// TwinCAT 3 PLC project Regions
// ProgramVersion: 3.1.4026.18
// libraries:
//   Tc3_Module, * (Beckhoff Automation GmbH)
//   ZApplication, 1.5.37.1 (Zeugwerk GmbH)
//   ZAux, 1.5.37.1 (Zeugwerk GmbH)
//   ZCore, 1.5.37.1 (Zeugwerk GmbH)
//   ZEquipment, 1.5.37.1 (Zeugwerk GmbH)
//   ZPlatform, 1.5.37.1 (Zeugwerk GmbH)
// project tree:
//   ZApp/App/ ZApp.TcPOU
//   ZApp/App/_DataTypes/ ZAppStep.TcDUT
//   ZApp/App/_States/ ZAppSequenceBoot.TcPOU, ZAppSequenceBootFault.TcPOU, ZAppSequenceRunning.TcPOU
//   ZApp/App/_SubObjects/ ZAppSequence.TcPOU
//   ZApp/Com/_DataTypes/ ZCom.TcDUT, ZComUnit.TcDUT
//   ZApp/Data/_DataTypes/ ZData.TcDUT, ZDataMachine.TcDUT, ZDataConfig.TcDUT, ZDataCalibration.TcDUT, ZDataRecipe.TcDUT
//   ZApp/SharedContext/ SharedContextCom.TcDUT, SharedContextComPublish.TcDUT, SharedContextComSubscribe.TcDUT, SharedContextContainer.TcPOU
//   ZApp/Unit/Handling/ HandlingUnit.TcPOU, HandlingUnitProgram.TcPOU, IHandling.TcIO
//   ZApp/Unit/Handling/_Com/ HandlingCom.TcDUT, HandlingComPublish.TcDUT, HandlingComPublishEquipment.TcDUT, HandlingComRef.TcDUT, HandlingComRequest.TcDUT, HandlingComSubscribe.TcDUT, HandlingComSubscribeEquipment.TcDUT
//   ZApp/Unit/Handling/_DataTypes/ HandlingState.TcDUT, HandlingStep.TcDUT
//   ZApp/Unit/Handling/_Data/ HandlingDataCalibration.TcDUT, HandlingDataConfig.TcDUT, HandlingDataMachine.TcDUT, HandlingDataRef.TcDUT
//   ZApp/Unit/Handling/_Equipment/ HandlingActuator.TcPOU, HandlingAxis.TcPOU, HandlingEquipment.TcPOU, HandlingFieldbus.TcPOU, HandlingIo.TcPOU, HandlingLinkedUnit.TcPOU
//   ZApp/Unit/Handling/_States/ HandlingSequenceAutomatic.TcPOU, HandlingSequenceBoot.TcPOU, HandlingSequenceFaultReaction.TcPOU, HandlingSequenceGoHome.TcPOU, HandlingSequenceStop.TcPOU, IPathQuery.TcIO, IPathQuery2.TcIO, IPathQuery3.TcIO, Path1d.TcPOU
//   ZApp/Unit/Handling/_SubObjects/ HandlingContainer.TcPOU, HandlingSequence.TcPOU
//   ZApp/ ZGlobal.TcGVL, ZModuleProgram.TcPOU, ZModuleTask.TcTTO
// real-time tasks:
//   TASK ZModuleTask: cycle T#10ms, priority 20, ADS port 350

CONFIGURATION Regions
    RESOURCE PLC ON TwinCAT3
        TASK ZModuleTask(INTERVAL := T#10ms, PRIORITY := 20);
        PROGRAM ZModuleProgram WITH ZModuleTask : ZModuleProgram;
    END_RESOURCE
END_CONFIGURATION

// ---- ZApp/App/_DataTypes/ZAppStep.TcDUT
{attribute 'qualified_only'}
{attribute 'to_string'}
TYPE ZAppStep :
(
  Undefined := 0
  
  ,BootBegin
  ,BootLoadDefaultData
  ,BootEnd
  ,BootFaultBegin
  ,BootFaultEnd 
  ,RunningBegin
  ,RunningEnd   
);
END_TYPE

// ---- ZApp/Com/_DataTypes/ZCom.TcDUT
TYPE ZCom :
STRUCT
  // module context
  App : ZApplication.ApplicationComPublish;
  Alarming : ZApplication.AlarmingCom;
  Messages : ZApplication.MessagingCom;
  
  // unit context
  Unit : ZComUnit;
  SharedContext : SharedContextCom;

END_STRUCT
END_TYPE

// ---- ZApp/Com/_DataTypes/ZComUnit.TcDUT
TYPE ZComUnit :
STRUCT
{region "Handling1"}
{IF NOT (defined (Handling1_disabled))}
  Handling1 : HandlingCom;
  {attribute 'ZId' := 'daa053b3-ae33-4567-9b11-72e6fc346262'}
{END_IF}
{endregion}
{region "Handling2"}
{IF NOT (defined (Handling2_disabled))}
  Handling2 : HandlingCom;
  {attribute 'ZId' := '686d4019-fd8f-49d1-bfb7-e2c5e589b8a3'}
{END_IF}
{endregion}
{region "Handling3"}
{IF NOT (defined (Handling3_disabled))}
  Handling3 : HandlingCom;
  {attribute 'ZId' := '12b42cce-14ce-45ff-90cd-901aacabced4'}
{END_IF}
{endregion}
{region "Handling4"}
{IF NOT (defined (Handling4_disabled))}
  Handling4 : HandlingCom;
  {attribute 'ZId' := '0a2dd986-966c-44be-a2b7-029bd083f361'}
{END_IF}
{endregion}
{attribute '__ZwPlcApplicationComUnitDeclaration__'} // Do not remove this attribute! It is used for code generation.
END_STRUCT
END_TYPE

// ---- ZApp/Data/_DataTypes/ZData.TcDUT
TYPE ZData :
STRUCT
  Config : ZDataConfig;
  Machine : ZDataMachine;
  Calibration : ZDataCalibration;
  Recipe : ZDataRecipe;
END_STRUCT
END_TYPE

// ---- ZApp/Data/_DataTypes/ZDataMachine.TcDUT
TYPE ZDataMachine :
STRUCT
{region "Handling1"}
{IF NOT (defined (Handling1_disabled))}
  Handling1 : HandlingDataMachine;
  {attribute 'ZId' := 'daa053b3-ae33-4567-9b11-72e6fc346262'}
{END_IF}
{endregion}
{region "Handling2"}
{IF NOT (defined (Handling2_disabled))}
  Handling2 : HandlingDataMachine;
  {attribute 'ZId' := '686d4019-fd8f-49d1-bfb7-e2c5e589b8a3'}
{END_IF}
{endregion}
{region "Handling3"}
{IF NOT (defined (Handling3_disabled))}
  Handling3 : HandlingDataMachine;
  {attribute 'ZId' := '12b42cce-14ce-45ff-90cd-901aacabced4'}
{END_IF}
{endregion}
{region "Handling4"}
{IF NOT (defined (Handling4_disabled))}
  Handling4 : HandlingDataMachine;
  {attribute 'ZId' := '0a2dd986-966c-44be-a2b7-029bd083f361'}
{END_IF}
{endregion}
{attribute '__ZwPlcApplicationDataMachineDeclaration__'} // Do not remove this attribute! It is used for code generation.
END_STRUCT
END_TYPE

// ---- ZApp/Data/_DataTypes/ZDataConfig.TcDUT
TYPE ZDataConfig :
STRUCT
{region "Handling1"}
{IF NOT (defined (Handling1_disabled))}
  Handling1 : HandlingDataConfig;
  {attribute 'ZId' := 'daa053b3-ae33-4567-9b11-72e6fc346262'}
{END_IF}
{endregion}
{region "Handling2"}
{IF NOT (defined (Handling2_disabled))}
  Handling2 : HandlingDataConfig;
  {attribute 'ZId' := '686d4019-fd8f-49d1-bfb7-e2c5e589b8a3'}
{END_IF}
{endregion}
{region "Handling3"}
{IF NOT (defined (Handling3_disabled))}
  Handling3 : HandlingDataConfig;
  {attribute 'ZId' := '12b42cce-14ce-45ff-90cd-901aacabced4'}
{END_IF}
{endregion}
{region "Handling4"}
{IF NOT (defined (Handling4_disabled))}
  Handling4 : HandlingDataConfig;
  {attribute 'ZId' := '0a2dd986-966c-44be-a2b7-029bd083f361'}
{END_IF}
{endregion}
{attribute '__ZwPlcApplicationDataConfigDeclaration__'} // Do not remove this attribute! It is used for code generation.
END_STRUCT
END_TYPE

// ---- ZApp/Data/_DataTypes/ZDataCalibration.TcDUT
TYPE ZDataCalibration :
STRUCT
{region "Handling1"}
{IF NOT (defined (Handling1_disabled))}
  Handling1 : HandlingDataCalibration;
  {attribute 'ZId' := 'daa053b3-ae33-4567-9b11-72e6fc346262'}
{END_IF}
{endregion}
{region "Handling2"}
{IF NOT (defined (Handling2_disabled))}
  Handling2 : HandlingDataCalibration;
  {attribute 'ZId' := '686d4019-fd8f-49d1-bfb7-e2c5e589b8a3'}
{END_IF}
{endregion}
{region "Handling3"}
{IF NOT (defined (Handling3_disabled))}
  Handling3 : HandlingDataCalibration;
  {attribute 'ZId' := '12b42cce-14ce-45ff-90cd-901aacabced4'}
{END_IF}
{endregion}
{region "Handling4"}
{IF NOT (defined (Handling4_disabled))}
  Handling4 : HandlingDataCalibration;
  {attribute 'ZId' := '0a2dd986-966c-44be-a2b7-029bd083f361'}
{END_IF}
{endregion}
{attribute '__ZwPlcApplicationDataCalibrationDeclaration__'} // Do not remove this attribute! It is used for code generation.
END_STRUCT
END_TYPE

// ---- ZApp/Data/_DataTypes/ZDataRecipe.TcDUT
TYPE ZDataRecipe :
STRUCT
  RecipeParam1 : LREAL;
  RecipeParam2 : LREAL;
  RecipeParam3 : LREAL;
END_STRUCT
END_TYPE

// ---- ZApp/SharedContext/SharedContextCom.TcDUT
TYPE SharedContextCom :
STRUCT
  Publish : SharedContextComPublish;
  Subscribe : SharedContextComSubscribe;
END_STRUCT
END_TYPE

// ---- ZApp/SharedContext/SharedContextComPublish.TcDUT
TYPE SharedContextComPublish :
STRUCT
  Region1 : ZApplication.RegionComPublish;
  Region2 : ZApplication.RegionComPublish;
  Region3 : ZApplication.RegionComPublish;
  Region4 : ZApplication.RegionComPublish;
  Region5 : ZApplication.RegionComPublish;
  Region6 : ZApplication.RegionComPublish;
  Region7 : ZApplication.RegionComPublish;
END_STRUCT
END_TYPE

// ---- ZApp/SharedContext/SharedContextComSubscribe.TcDUT
TYPE SharedContextComSubscribe :
STRUCT
  Region1 : ZApplication.RegionComSubscribe;
  Region2 : ZApplication.RegionComSubscribe;
  Region3 : ZApplication.RegionComSubscribe;
  Region4 : ZApplication.RegionComSubscribe;
  Region5 : ZApplication.RegionComSubscribe;
  Region6 : ZApplication.RegionComSubscribe;
  Region7 : ZApplication.RegionComSubscribe;
END_STRUCT
END_TYPE

// ---- ZApp/Unit/Handling/_Com/HandlingCom.TcDUT
/// This struct contains variables that
/// * are read from outside (e.g. HMI) to retrieve information about the unit's current state and (temporary) parameters (= `publish`) 
/// * are written from outside (e.g. HMI) to control the unit via ADS (= `subscribe`) 
TYPE HandlingCom :
STRUCT
  Publish : HandlingComPublish;
  Subscribe : HandlingComSubscribe;
END_STRUCT
END_TYPE

// ---- ZApp/Unit/Handling/_Com/HandlingComPublish.TcDUT
/// this is the container of informations that the unit wants to share with the world outside of the PLC
/// This struct should only be read from by external applications.
TYPE HandlingComPublish :
STRUCT
  State : ZApplication.UnitStateMachineState; // state the unit is in
  Request : HandlingComRequest; // booleans that indictate which action is currently possible to perform with this unit
  Equipment : HandlingComPublishEquipment;  // structs for equipment objects which are used by the bridges
  
  TargetPosition : LREAL;
END_STRUCT
END_TYPE

// ---- ZApp/Unit/Handling/_Com/HandlingComPublishEquipment.TcDUT
TYPE HandlingComPublishEquipment :
STRUCT

{region "AxisX : Axis"}
  AxisX : ZApplication.AxisComPublish;
  {attribute 'ZId' := '948ae39b-c3c7-40c3-a820-f277405d18e6'}
{endregion}

{attribute '__ZwPlcUnitComDeclaration__'} // Do not remove this attribute! It is used for code generation.

END_STRUCT
END_TYPE

// ---- ZApp/Unit/Handling/_Com/HandlingComRef.TcDUT
/// container for all communication data types that are used by the unit
TYPE HandlingComRef :
STRUCT
  Publish : REFERENCE TO HandlingComPublish; 
  Subscribe : REFERENCE TO HandlingComSubscribe; 
END_STRUCT
END_TYPE

// ---- ZApp/Unit/Handling/_Com/HandlingComRequest.TcDUT
TYPE HandlingComRequest :
STRUCT
  Start : BOOL;
  Stop : BOOL;
  GoHome : BOOL;
  Halt : BOOL;
END_STRUCT
END_TYPE

// ---- ZApp/Unit/Handling/_Com/HandlingComSubscribe.TcDUT
TYPE HandlingComSubscribe :
STRUCT
  Request : HandlingComRequest; // contains booleans that are used to start a specific sequence.
  Equipment : HandlingComSubscribeEquipment;  // structs for equipment objects which are used by the bridges
END_STRUCT
END_TYPE

// ---- ZApp/Unit/Handling/_Com/HandlingComSubscribeEquipment.TcDUT
TYPE HandlingComSubscribeEquipment :
STRUCT

{region "AxisX : Axis"}
  AxisX : ZApplication.AxisComSubscribe;
  {attribute 'ZId' := '948ae39b-c3c7-40c3-a820-f277405d18e6'}
{endregion}

{attribute '__ZwPlcUnitComDeclaration__'} // Do not remove this attribute! It is used for code generation.

END_STRUCT
END_TYPE

// ---- ZApp/Unit/Handling/_DataTypes/HandlingState.TcDUT
/// This enumeration contains all used defined sequences of a unit.
/// Per default a unit makes use of the states that are contained in (UnitStateDefault)[xref:ZApplication.UnitStateDefault]. However,
/// most of the time a unit need to perform some application depend sequences that can be performed by putting the unit into userdefined states.
/// For instance, a robotic unit could use the state (automatic)[xref:ZApplication.UnitStateDefault] to lift an object from point A to point B,
/// a userdefined state could be used to open and close the robotic-units gripper, respectively
{attribute 'qualified_only'}
TYPE HandlingState :
(
	UserdefinedState1 := ZApplication.UnitStateMachineState.Last+1
);
END_TYPE

// ---- ZApp/Unit/Handling/_DataTypes/HandlingStep.TcDUT
/// This enumeration contains all steps that are used by the various sequences of a unit.
/// Sequences use a subrange (***Begin to ***End) of this enumeration.
{attribute 'qualified_only'}
{attribute 'to_string'}
TYPE HandlingStep :
(
  Undefined := 0
  
  ,BootBegin
  ,BootEnd 

  ,StopBegin
  ,StopEnd

  ,AutomaticBegin
  ,AutomaticWait
  ,AutomaticReservePath
  ,AutomaticMoveThroughRegion
  ,AutomaticMoveToEndPosition
  ,AutomaticMove
  ,AutomaticEnd
  
  ,GoHomeBegin
  ,GoHomeEnd 
  
  ,FaultReactionBegin
  ,FaultReactionEnd
);
END_TYPE

// ---- ZApp/Unit/Handling/_Data/HandlingDataCalibration.TcDUT
/// calibration that is determined by calibration sequences of the unit (static offsets, shifts)
TYPE HandlingDataCalibration :
STRUCT
END_STRUCT
END_TYPE

// ---- ZApp/Unit/Handling/_Data/HandlingDataConfig.TcDUT
/// configuration data that is used during boot to configure the Units equipment
TYPE HandlingDataConfig :
STRUCT
  Simulated : BOOL;
END_STRUCT
END_TYPE

// ---- ZApp/Unit/Handling/_Data/HandlingDataMachine.TcDUT
/// machine data that is used through most sequences of the unit (motor speed, axes positions, ...)
TYPE HandlingDataMachine :
STRUCT
  Slowspeed : LREAL;
  Highspeed : LREAL;
END_STRUCT
END_TYPE

// ---- ZApp/Unit/Handling/_Data/HandlingDataRef.TcDUT
/// container for all data that are used by the unit
TYPE HandlingDataRef :
STRUCT
  Config : REFERENCE TO HandlingDataConfig; // data required for booting the unit (axes configuration, simulation, parameters that have to be written in PREOP, ...)
  Machine : REFERENCE TO HandlingDataMachine; // speeds, positions, ...
  Calibration : REFERENCE TO HandlingDataCalibration; // offsets, shifts of nominal to actual values
END_STRUCT
END_TYPE

// ---- ZApp/ZGlobal.TcGVL
{attribute 'qualified_only'}
VAR_GLOBAL
  Com : ZCom;
END_VAR
VAR_GLOBAL PERSISTENT
  Data : ZData;
END_VAR

// ---- ZApp/Unit/Handling/IHandling.TcIO
INTERFACE IHandling EXTENDS ZApplication.IUnit

END_INTERFACE

// ---- ZApp/Unit/Handling/_States/IPathQuery.TcIO
INTERFACE IPathQuery

METHOD FromPosition : IPathQuery2
VAR_INPUT
  pos : LREAL;
END_VAR
END_METHOD

METHOD WithSafetyMargin : IPathQuery
VAR_INPUT
  margin : LREAL;
END_VAR
END_METHOD

METHOD WithSortedRegions : IPathQuery
VAR_INPUT
  regions : POINTER TO ZApplication.Region;
  regionCount : INT;
END_VAR
END_METHOD

METHOD WithWidth : IPathQuery
VAR_INPUT
  width : LREAL;
END_VAR
END_METHOD

END_INTERFACE

// ---- ZApp/Unit/Handling/_States/IPathQuery2.TcIO
INTERFACE IPathQuery2

METHOD ToPosition : IPathQuery3
VAR_INPUT
  pos : LREAL;
END_VAR
END_METHOD

END_INTERFACE

// ---- ZApp/Unit/Handling/_States/IPathQuery3.TcIO
INTERFACE IPathQuery3

METHOD ReserveAsync
VAR_INPUT
  unit : REFERENCE TO Unit;
END_VAR
END_METHOD

END_INTERFACE

// ---- ZApp/ZModuleProgram.TcPOU
/// Zeugwerk Application
PROGRAM ZModuleProgram
VAR_INPUT
{region "ZModuleProgram : Utility"}
  App : ZApp(displayName:='Zeugwerk-Application Template', com:=ZGlobal.Com.App);
  Datetime : ZAux.DateTimeUM;
  {attribute 'ZId' := ''}
{endregion}
{region "ZModuleProgram : Logging"}
  Alarming : ZApplication.Alarming(App, datetime := Datetime, com := ZGlobal.Com.Alarming);
  LoggerHmi : ZApplication.Messaging(App, datetime := Datetime, com := ZGlobal.Com.Messages);
  LoggerFile : ZAux.LoggerFile7FF(App, datetime := Datetime, filePath:='C:\Zeugwerk\logs\messages.log', target:='');
  Logger : ZAux.Logging;
  {attribute 'ZId' := ''}
{endregion}  
{attribute '__ZwPlcApplicationModuleProgramDeclaration__'} // Do not remove this attribute! It is used for code generation.
  SharedContext : SharedContextContainer(parent := App, com := ZGlobal.Com.SharedContext, logger := Logger);
{region "Handling1"}
{undefine RunInSeparateProgram}
{IF NOT (defined (Handling1_disabled)) AND NOT (defined (RunInSeparateProgram))}
  Handling1 : HandlingUnit(displayName := 'Handling1', // name of the unit (for logging)
    parent:= App,
    configdata:= ZGlobal.Data.Config.Handling1,
    machinedata := ZGlobal.Data.Machine.Handling1,
    calibrationdata := ZGlobal.Data.Calibration.Handling1,
    com := ZGlobal.Com.Unit.Handling1,
    logger := Logger,
    alarming:= Alarming);
  {attribute 'section' := '__ZwPlcUnitProgramDeclaration__'}
  {attribute 'ZId' := 'daa053b3-ae33-4567-9b11-72e6fc346262'}
{END_IF}
{endregion}
{region "Handling2"}
{undefine RunInSeparateProgram}
{IF NOT (defined (Handling2_disabled)) AND NOT (defined (RunInSeparateProgram))}
  Handling2 : HandlingUnit(displayName := 'Handling2', // name of the unit (for logging)
    parent:= App,
    configdata:= ZGlobal.Data.Config.Handling2,
    machinedata := ZGlobal.Data.Machine.Handling2,
    calibrationdata := ZGlobal.Data.Calibration.Handling2,
    com := ZGlobal.Com.Unit.Handling2,
    logger := Logger,
    alarming:= Alarming);
  {attribute 'section' := '__ZwPlcUnitProgramDeclaration__'}
  {attribute 'ZId' := '686d4019-fd8f-49d1-bfb7-e2c5e589b8a3'}
{END_IF}
{endregion}
{region "Handling3"}
{undefine RunInSeparateProgram}
{IF NOT (defined (Handling3_disabled)) AND NOT (defined (RunInSeparateProgram))}
  Handling3 : HandlingUnit(displayName := 'Handling3', // name of the unit (for logging)
    parent:= App,
    configdata:= ZGlobal.Data.Config.Handling3,
    machinedata := ZGlobal.Data.Machine.Handling3,
    calibrationdata := ZGlobal.Data.Calibration.Handling3,
    com := ZGlobal.Com.Unit.Handling3,
    logger := Logger,
    alarming:= Alarming);
  {attribute 'section' := '__ZwPlcUnitProgramDeclaration__'}
  {attribute 'ZId' := '12b42cce-14ce-45ff-90cd-901aacabced4'}
{END_IF}
{endregion}
{region "Handling4"}
{undefine RunInSeparateProgram}
{IF NOT (defined (Handling4_disabled)) AND NOT (defined (RunInSeparateProgram))}
  Handling4 : HandlingUnit(displayName := 'Handling4', // name of the unit (for logging)
    parent:= App,
    configdata:= ZGlobal.Data.Config.Handling4,
    machinedata := ZGlobal.Data.Machine.Handling4,
    calibrationdata := ZGlobal.Data.Calibration.Handling4,
    com := ZGlobal.Com.Unit.Handling4,
    logger := Logger,
    alarming:= Alarming);
  {attribute 'section' := '__ZwPlcUnitProgramDeclaration__'}
  {attribute 'ZId' := '0a2dd986-966c-44be-a2b7-029bd083f361'}
{END_IF}
{endregion}
{attribute '__ZwPlcUnitProgramDeclaration__'} // Do not remove this attribute! It is used for code generation.
END_VAR

{region "ZModuleProgram : Utility"}
  Datetime.Cyclic();
  App.Cyclic();
  {attribute 'ZId' := ''}
{endregion}
{attribute '__ZwPlcApplicationModuleProgramImplementation__'} // Do not remove this attribute! It is used for code generation.

END_PROGRAM

// ---- ZApp/App/ZApp.TcPOU
FUNCTION_BLOCK ZApp EXTENDS ZApplication.Application
VAR
  _boot : ZAppSequenceBoot;
  _bootFault : ZAppSequenceBootFault;
  _running : ZAppSequenceRunning;
END_VAR

METHOD FB_init : BOOL
VAR_INPUT
  bInitRetains : BOOL; /// if TRUE, the retain variables are initialized (warm start / cold start)
  bInCopyCode : BOOL; /// if TRUE, the instance afterwards gets moved into the copy code (online change)
  displayName : ZCore.ZString;
  com : REFERENCE TO ZApplication.ApplicationComPublish;
END_VAR
SetBootSequence(_boot);
SetBootFaultSequence(_bootFault);
SetRunningSequence(_running);
END_METHOD

END_FUNCTION_BLOCK

// ---- ZApp/App/_States/ZAppSequenceBoot.TcPOU
FUNCTION_BLOCK ZAppSequenceBoot EXTENDS ZAppSequence IMPLEMENTS ZCore.ISequence
VAR
  _step : ZCore.Step(ZAppStep.BootBegin, ZAppStep.BootEnd);
END_VAR

IF OnStart(_step)
THEN
  // init custom sequence variables here ...
END_IF

REPEAT
  LogStep();

  CASE _step.Index OF
    (* -------------------------------------------------------------------------------------------------------------------------------- *)
    ZAppStep.BootBegin:
    (* -------------------------------------------------------------------------------------------------------------------------------- *)
    
      IF _step.OnEntry()
      THEN
        ZModuleProgram.LoggerFile.MinimumLevel := ZCore.LogLevel.Trace;
        ZModuleProgram.Logger.AddLogger(ZModuleProgram.LoggerFile);        
        {attribute '__ZwPlcAppZComModuleContext__'} // Do not remove this attribute! It is used for code generation.      
      END_IF
      
	  IF ZModuleProgram.Datetime.State <> ZCore.ObjectState.Booting
      THEN
        _step.SetNext(ZAppStep.BootLoadDefaultData);        
      END_IF
      
    (* -------------------------------------------------------------------------------------------------------------------------------- *)
    ZAppStep.BootLoadDefaultData:
    (* -------------------------------------------------------------------------------------------------------------------------------- *)

      {warning 'The application is loading the default config data on every restart!'}
      LoadDefaultConfigData();
      ZModuleProgram.SharedContext();
      
      IF IsCommissioning()
      THEN
        LoadDefaultData();
      END_IF
      
      _step.SetNext(ZAppStep.BootEnd);
      
    (* -------------------------------------------------------------------------------------------------------------------------------- *)
    ZAppStep.BootEnd:
    (* -------------------------------------------------------------------------------------------------------------------------------- *)
      SetBusy(FALSE);
      
  ELSE
    Abort('sequence contains unhandled step');
  END_CASE
UNTIL _step.IsNotRepeatable() OR_ELSE NOT Busy END_REPEAT

METHOD  IsCommissioning : BOOL
IsCommissioning := TRUE;
END_METHOD

METHOD FINAL LoadDefaultConfigData

{region "Handling1"}
  {IF NOT (defined (Handling1_disabled))}
  ZGlobal.Data.Config.Handling1.Simulated := TRUE;
  {region "UserInitCode"}
  // put your individual init code for this unit here
  {endregion}
  {END_IF}
  {attribute 'ZId' := 'daa053b3-ae33-4567-9b11-72e6fc346262'}
{endregion}

{region "Handling2"}
  {IF NOT (defined (Handling2_disabled))}
  ZGlobal.Data.Config.Handling2.Simulated := TRUE;
  {region "UserInitCode"}
  // put your individual init code for this unit here
  {endregion}
  {END_IF}
  {attribute 'ZId' := '686d4019-fd8f-49d1-bfb7-e2c5e589b8a3'}
{endregion}

{region "Handling3"}
  {IF NOT (defined (Handling3_disabled))}
  ZGlobal.Data.Config.Handling3.Simulated := TRUE;
  {region "UserInitCode"}
  // put your individual init code for this unit here
  {endregion}
  {END_IF}
  {attribute 'ZId' := '12b42cce-14ce-45ff-90cd-901aacabced4'}
{endregion}

{region "Handling4"}
  {IF NOT (defined (Handling4_disabled))}
  ZGlobal.Data.Config.Handling4.Simulated := TRUE;
  {region "UserInitCode"}
  // put your individual init code for this unit here
  {endregion}
  {END_IF}
  {attribute 'ZId' := '0a2dd986-966c-44be-a2b7-029bd083f361'}
{endregion}

{attribute '__ZwPlcUnitLoadDefaultConfigData__'} // Do not remove this attribute! It is used for code generation.
END_METHOD

METHOD FINAL LoadDefaultData

{attribute '__ZwPlcUnitLoadDefaultData__'} // Do not remove this attribute! It is used for code generation.
END_METHOD

END_FUNCTION_BLOCK

// ---- ZApp/App/_SubObjects/ZAppSequence.TcPOU
FUNCTION_BLOCK ABSTRACT ZAppSequence EXTENDS ZApplication.Sequence IMPLEMENTS ZCore.ISequence

METHOD StepDecoded : ZCore.ZString
VAR_INPUT
  stepIndex : INT;
END_VAR
VAR_INST
  _stepIndexDecoded : ZAppStep;
END_VAR
_stepIndexDecoded := stepIndex;
StepDecoded := TO_STRING(_stepIndexDecoded);
END_METHOD

END_FUNCTION_BLOCK

// ---- ZApp/App/_States/ZAppSequenceBootFault.TcPOU
FUNCTION_BLOCK ZAppSequenceBootFault EXTENDS ZAppSequence IMPLEMENTS ZCore.ISequence
VAR
  _step : ZCore.Step(ZAppStep.BootFaultBegin, ZAppStep.BootFaultEnd);
END_VAR

IF OnStart(_step)
THEN
  // init custom sequence variables here ...
END_IF

REPEAT
  LogStep();

  CASE _step.Index OF
    (* -------------------------------------------------------------------------------------------------------------------------------- *)
    ZAppStep.BootFaultBegin:
    (* -------------------------------------------------------------------------------------------------------------------------------- *)
      _step.SetNext(ZAppStep.BootFaultEnd);
      
    (* -------------------------------------------------------------------------------------------------------------------------------- *)
    ZAppStep.BootFaultEnd:
    (* -------------------------------------------------------------------------------------------------------------------------------- *)
      SetBusy(FALSE);
      
  ELSE
    Abort('sequence contains unhandled step');
  END_CASE
UNTIL _step.IsNotRepeatable() OR_ELSE NOT Busy END_REPEAT

END_FUNCTION_BLOCK

// ---- ZApp/App/_States/ZAppSequenceRunning.TcPOU
FUNCTION_BLOCK ZAppSequenceRunning EXTENDS ZAppSequence IMPLEMENTS ZCore.ISequence
VAR
  _step : ZCore.Step(ZAppStep.RunningBegin, ZAppStep.RunningEnd);
END_VAR

IF OnStart(_step)
THEN
  // init custom sequence variables here ...
END_IF

REPEAT
  LogStep();

  CASE _step.Index OF
    (* -------------------------------------------------------------------------------------------------------------------------------- *)
    ZAppStep.RunningBegin:
    (* -------------------------------------------------------------------------------------------------------------------------------- *)
      ; // implement me
      
    (* -------------------------------------------------------------------------------------------------------------------------------- *)
    ZAppStep.RunningEnd:
    (* -------------------------------------------------------------------------------------------------------------------------------- *)
      SetBusy(FALSE);
      
  ELSE
    Abort('sequence contains unhandled step');
  END_CASE
UNTIL _step.IsNotRepeatable() OR_ELSE NOT Busy END_REPEAT

END_FUNCTION_BLOCK

// ---- ZApp/SharedContext/SharedContextContainer.TcPOU
FUNCTION_BLOCK SharedContextContainer EXTENDS ZCore.ObjectContainer
VAR_INPUT
  Region1 : ZApplication.Region('Region-1', priority:=13);
  Region2 : ZApplication.Region('Region-2', priority:=12);
  Region3 : ZApplication.Region('Region-3', priority:=11);  
  Region4 : ZApplication.Region('Region-4', priority:=4);  
  Region5 : ZApplication.Region('Region-5', priority:=5);  
  Region6 : ZApplication.Region('Region-6', priority:=6);  
  Region7 : ZApplication.Region('Region-7', priority:=7);  

  
END_VAR
VAR
  {attribute 'hide'}
  _regionbridge : ZApplication.RegionBridge(0);  
  _logger : ZCore.ILogger;
  _com : REFERENCE TO SharedContextCom;  
  v1, v2 : ZCore.Vector4;
END_VAR

IF _isInitialized
THEN
  RETURN;
END_IF

v1.Y := -25;
v2.Y := 25;

v1.X := 100;
v2.X := 150;
Region1.SetBoundingBox(v1, v2);
Region1.SetLogger(_logger);
_regionbridge.AddStaticRegion(Region1, _com.Publish.Region1, _com.Subscribe.Region1);

v1.X := 250;
v2.X := 300;
Region2.SetBoundingBox(v1, v2);
Region2.SetLogger(_logger);
_regionbridge.AddStaticRegion(Region2, _com.Publish.Region2, _com.Subscribe.Region2);

v1.X := 305;
v2.X := 355;
Region3.SetBoundingBox(v1, v2);
Region3.SetLogger(_logger);
_regionbridge.AddStaticRegion(Region3, _com.Publish.Region3, _com.Subscribe.Region3);

v1.X := 360;
v2.X := 410;
Region4.SetBoundingBox(v1, v2);
Region4.SetLogger(_logger);
_regionbridge.AddStaticRegion(Region4, _com.Publish.Region4, _com.Subscribe.Region4);


v1.X := 480;
v2.X := 530;
Region5.SetBoundingBox(v1, v2);
Region5.SetLogger(_logger);
_regionbridge.AddStaticRegion(Region5, _com.Publish.Region5, _com.Subscribe.Region5);


v1.X := 650;
v2.X := 700;
Region6.SetBoundingBox(v1, v2);
Region6.SetLogger(_logger);
_regionbridge.AddStaticRegion(Region6, _com.Publish.Region6, _com.Subscribe.Region6);


v1.X := 705;
v2.X := 755;
Region7.SetBoundingBox(v1, v2);
Region7.SetLogger(_logger);
_regionbridge.AddStaticRegion(Region7, _com.Publish.Region7, _com.Subscribe.Region7);


_isInitialized := TRUE;

//FB_Init is always available implicitly and it is used primarily for initialization.
//The return value is not evaluated. For a specific influence, you can also declare the
//methods explicitly and provide additional code there with the standard initialization
//code. You can evaluate the return value.
METHOD FB_Init: BOOL
VAR_INPUT
  bInitRetains: BOOL; // TRUE: the retain variables are initialized (reset warm / reset cold)
  bInCopyCode: BOOL;  // TRUE: the instance will be copied to the copy code afterward (online change)
  parent : ZCore.IManagedObject;
  com : REFERENCE TO SharedContextCom;
  logger : ZCore.ILogger;
END_VAR
_logger := logger;
_com REF= com;
_regionbridge.FB_init(bInitRetains, bInCopyCode, parent);
END_METHOD

END_FUNCTION_BLOCK

// ---- ZApp/Unit/Handling/HandlingUnit.TcPOU
FUNCTION_BLOCK HandlingUnit EXTENDS ZApplication.Unit IMPLEMENTS IHandling
VAR
  _equipment : HandlingEquipment(THIS^);
  _data : HandlingDataRef;
  _com : HandlingComRef;

  _boot : HandlingSequenceBoot(THIS^);
  _automatic : HandlingSequenceAutomatic(THIS^);
  _stop : HandlingSequenceStop(THIS^);
  _gohome : HandlingSequenceGoHome(THIS^);
  _faultReaction : HandlingSequenceFaultReaction(THIS^);
  
  _statemachine : ZApplication.UnitStateMachine;

  _observeTimer : ZAux.Timer;
END_VAR

{attribute 'ZId' := '19816701-366b-4384-b6ea-ebe33b677430'}

IF _statemachine.State() = ZApplication.UnitStateMachineState.Automatic
THEN
  _com.Publish.TargetPosition := _automatic.CurrentTargetPosition;
ELSE
  _com.Publish.TargetPosition := _equipment.Axis.AxisX.ActualPosition;
END_IF

IF _observeTimer.Done THEN
  _observeTimer.WaitAsync(0.1);
  
  // monitor _com for requested actions (e.g. start homing, start automatic mode, ...)
  ObserveRequest(_com.Subscribe.Request.Start, ZApplication.UnitStateMachineState.Automatic);
  ObserveRequest(_com.Subscribe.Request.Stop, ZApplication.UnitStateMachineState.Stop);
  ObserveRequest(_com.Subscribe.Request.GoHome, ZApplication.UnitStateMachineState.GoHome);
  ObserveRequest(_com.Subscribe.Request.Halt, ZApplication.UnitStateMachineState.Halt);
  
  // provide relevant information via ADS
  _com.Publish.Request.Stop := _stateMachine.IsTransitionAllowed(ZApplication.UnitStateMachineState.Stop);
  _com.Publish.Request.Start := _stateMachine.IsTransitionAllowed(ZApplication.UnitStateMachineState.Automatic);
  _com.Publish.Request.GoHome := _stateMachine.IsTransitionAllowed(ZApplication.UnitStateMachineState.GoHome);
  _com.Publish.Request.Halt := _stateMachine.IsTransitionAllowed(ZApplication.UnitStateMachineState.Halt);

  _com.Publish.State := _stateMachine.State();
END_IF

METHOD FB_init : BOOL
VAR_INPUT
  bInitRetains : BOOL;
  bInCopyCode : BOOL;
  parent : ZCore.IManagedObject;
  displayName : ZCore.ZString;
  configdata : REFERENCE TO HandlingDataConfig;
  machinedata : REFERENCE TO HandlingDataMachine;
  calibrationdata : REFERENCE TO HandlingDataCalibration;
  com : REFERENCE TO HandlingCom;
  logger : ZCore.ILogger;
  alarming: ZApplication.IAlarming;
END_VAR
_name := displayName;

// initialize local logger decorator
_loggerDecorator.FB_init(bInitRetains, bInCopyCode, _name, logger);
_alarmingDecorator.FB_init(bInitRetains, bInCopyCode, _name, alarming);

// setup data
_data.Config REF= configdata;
_data.Machine REF= machinedata;
_data.Calibration REF= calibrationdata;
_com.Publish REF= com.Publish;
_com.Subscribe REF= com.Subscribe;

// ------- sequence initialization, map sequences of this unit to the statemachine -------
{attribute '__ZwPlcUnitInitSequenceImplementation__'} // Do not remove this attribute! It is used for code generation.
_statemachine.SetSequence(ZApplication.UnitStateMachineState.Boot, _boot);
_statemachine.SetSequence(ZApplication.UnitStateMachineState.FaultReaction, _faultReaction);
_statemachine.SetSequence(ZApplication.UnitStateMachineState.Gohome, _gohome);
_statemachine.SetSequence(ZApplication.UnitStateMachineState.Stop, _stop);
_statemachine.SetSequence(ZApplication.UnitStateMachineState.Automatic, _automatic);

_statemachine.SetName(_name);
_statemachine.SetLogger(_logger);

// set initial state
_statemachine.SetState(ZApplication.UnitStateMachineState.Boot);
SetStateMachine(_statemachine);
END_METHOD

END_FUNCTION_BLOCK

// ---- ZApp/Unit/Handling/_Equipment/HandlingEquipment.TcPOU
/// This function block is a container for equipment that is used by this unit.
/// Equipment is grouped by its kind (actuator, axes, io, ...).
/// It extends from [ManagedObjectContainer](xref:ZCore.ManagedObjectContainer) such that the parent
/// (= the unit itself) can be passed to equipment instances.
FUNCTION_BLOCK HandlingEquipment EXTENDS HandlingContainer
VAR_INPUT
  Io : HandlingIo(_parent);
  Actuator : HandlingActuator(_parent);
  Axis : HandlingAxis(_parent);
  Fieldbus : HandlingFieldbus(_parent);
  Unit : HandlingLinkedUnit(_parent);
END_VAR

END_FUNCTION_BLOCK

// ---- ZApp/Unit/Handling/_SubObjects/HandlingContainer.TcPOU
FUNCTION_BLOCK HandlingContainer EXTENDS ZCore.ObjectContainer
VAR_INPUT
END_VAR
VAR_OUTPUT
END_VAR
VAR
  {attribute 'hide'}
  _parent : REFERENCE TO HandlingUnit;
END_VAR

{attribute 'hide' }
METHOD FB_init : BOOL
VAR_INPUT
	bInitRetains : BOOL; // if TRUE, the retain variables are initialized (warm start / cold start)
	bInCopyCode : BOOL;  // if TRUE, the instance afterwards gets moved into the copy code (online change)
  unit : REFERENCE TO HandlingUnit;
END_VAR
_parent REF= unit;
END_METHOD

END_FUNCTION_BLOCK

// ---- ZApp/Unit/Handling/_Equipment/HandlingIo.TcPOU
/// This function block is a container for all I/Os that are used by this unit.
/// The parent of all objects can be directly transfered in their constructor (this is only relevant for equipment objects
/// that have to be managed (e.g. [DebouncedInput](xref:ZEquipment.DebouncedInput), [Light](xref:ZEquipment.Light), ...).
FUNCTION_BLOCK HandlingIo EXTENDS HandlingContainer
VAR
  {attribute 'hide'}
  _iobridge : ZApplication.IoBridge(_parent);
END_VAR
VAR_INPUT

{attribute '__ZwPlcUnitEquipmentDeclaration__'} // Do not remove this attribute! It is used for code generation.
END_VAR

IF _isInitialized
THEN
  RETURN;
END_IF

  _iobridge.SetLogger(_parent._logger);

{attribute '__ZwPlcUnitEquipmentImplementation__'} // Do not remove this attribute! It is used for code generation.

_isInitialized := TRUE;

END_FUNCTION_BLOCK

// ---- ZApp/Unit/Handling/_Equipment/HandlingActuator.TcPOU
/// This function block is a container for all actuator objects that are used by this unit.
/// The parent of all objects can be directly transfered in their constructor (this is only relevant for equipment objects
/// that have to be managed (e.g. [DebouncedInput](xref:ZEquipment.DebouncedInput), [Light](xref:ZEquipment.Light), ...).
FUNCTION_BLOCK HandlingActuator EXTENDS HandlingContainer
VAR
  {attribute 'hide'}
  _actuatorbridge : ZApplication.ActuatorBridge(_parent);
  {attribute 'hide'}
  _iobridge : ZApplication.IoBridge(_parent);
END_VAR
VAR_INPUT

{attribute '__ZwPlcUnitEquipmentDeclaration__'} // Do not remove this attribute! It is used for code generation.
END_VAR

IF _isInitialized
THEN
  RETURN;
END_IF

  _actuatorbridge.SetLogger(_parent._logger);

{attribute '__ZwPlcUnitEquipmentImplementation__'} // Do not remove this attribute! It is used for code generation.

_isInitialized := TRUE;

END_FUNCTION_BLOCK

// ---- ZApp/Unit/Handling/_Equipment/HandlingAxis.TcPOU
/// This function block is a container for all axis objects that are used by this unit.
/// The parent of all objects can be directly transfered in their constructor (this is only relevant for equipment objects
/// that have to be managed (e.g. [DebouncedInput](xref:ZEquipment.DebouncedInput), [Light](xref:ZEquipment.Light), ...).
FUNCTION_BLOCK HandlingAxis EXTENDS HandlingContainer
VAR
  {attribute 'hide'}
  _axisbridge : ZApplication.AxisBridge(_parent);
END_VAR
VAR_INPUT

{region "AxisX : AxisPlcOpenMc"}
  AxisX : ZEquipment.AxisPlcOpenMc(_parent);
  {attribute 'ZId' := '948ae39b-c3c7-40c3-a820-f277405d18e6'}
{endregion}

{attribute '__ZwPlcUnitEquipmentDeclaration__'} // Do not remove this attribute! It is used for code generation.
END_VAR

IF _isInitialized
THEN
  RETURN;
END_IF

  _axisbridge.SetLogger(_parent._logger);

{region "AxisX : AxisPlcOpenMc"}
  AxisX.SetLogger(_parent._logger);
  AxisX.SetName(name:='AxisX');
  AxisX.SetSimulation(_parent._data.Config.Simulated);
  _axisbridge.AddAxisPlcOpenMc(axis:=AxisX, publish:=_parent._com.Publish.Equipment.AxisX, subscribe:=_parent._com.Subscribe.Equipment.AxisX);

  {region "UserInitCode"}
  // put your individual init code for this Axis here
  {endregion}

  {attribute 'ZId' := '948ae39b-c3c7-40c3-a820-f277405d18e6'}
{endregion}

{attribute '__ZwPlcUnitEquipmentImplementation__'} // Do not remove this attribute! It is used for code generation.

_isInitialized := TRUE;

END_FUNCTION_BLOCK

// ---- ZApp/Unit/Handling/_Equipment/HandlingFieldbus.TcPOU
/// This function block is a container for all axis objects that are used by this unit.
/// The parent of all objects can be directly transfered in their constructor (this is only relevant for equipment objects
/// that have to be managed (e.g. [DebouncedInput](xref:ZEquipment.DebouncedInput), [Light](xref:ZEquipment.Light), ...).
FUNCTION_BLOCK HandlingFieldbus EXTENDS HandlingContainer
VAR
END_VAR
VAR_INPUT

{attribute '__ZwPlcUnitEquipmentDeclaration__'} // Do not remove this attribute! It is used for code generation.
END_VAR

IF _isInitialized
THEN
  RETURN;
END_IF

{attribute '__ZwPlcUnitEquipmentImplementation__'} // Do not remove this attribute! It is used for code generation.

_isInitialized := TRUE;

END_FUNCTION_BLOCK

// ---- ZApp/Unit/Handling/_Equipment/HandlingLinkedUnit.TcPOU
/// This function block is a container for all linked units that are used by this unit.
/// Linked units can be addressed through their individual interface.
FUNCTION_BLOCK HandlingLinkedUnit EXTENDS HandlingContainer
VAR_INPUT

{attribute '__ZwPlcUnitEquipmentDeclaration__'} // Do not remove this attribute! It is used for code generation.
END_VAR

IF _isInitialized
THEN
  RETURN;
END_IF

{attribute '__ZwPlcUnitEquipmentImplementation__'} // Do not remove this attribute! It is used for code generation.

_isInitialized := TRUE;

END_FUNCTION_BLOCK

// ---- ZApp/Unit/Handling/_States/HandlingSequenceBoot.TcPOU
FUNCTION_BLOCK HandlingSequenceBoot EXTENDS HandlingSequence IMPLEMENTS ZCore.ISequence
VAR
  _step : ZCore.Step(HandlingStep.BootBegin, HandlingStep.BootEnd);
END_VAR

IF OnStart(_step) THEN
  ; // init custom sequence variables here ...
END_IF

REPEAT
  LogStep();

  CASE _step.Index OF
    (* -------------------------------------------------------------------------------------------------------------------------------- *)
    HandlingStep.BootBegin:
    (* -------------------------------------------------------------------------------------------------------------------------------- *)
      IF _step.OnEntry()
      THEN
        // initialize equipment
        _io();
        _actuator();
        _fieldbus();
        _axis();
        _unit();
      END_IF
      
      _parent._objectManager.Cyclic();      
      Assert(_parent._objectManager);
      IF _parent._objectManager.Booted
      THEN
        _step.SetNext(HandlingStep.BootEnd);
      END_IF

    (* -------------------------------------------------------------------------------------------------------------------------------- *)
    HandlingStep.BootEnd:
    (* -------------------------------------------------------------------------------------------------------------------------------- *)
      SetBusy(FALSE);
      
  ELSE
    Abort('sequence contains unhandled step');
  END_CASE
UNTIL _step.IsNotRepeatable() OR_ELSE NOT Busy END_REPEAT

END_FUNCTION_BLOCK

// ---- ZApp/Unit/Handling/_SubObjects/HandlingSequence.TcPOU
FUNCTION_BLOCK HandlingSequence EXTENDS ZApplication.Sequence
VAR
  {attribute 'hide'}
  _parent : REFERENCE TO HandlingUnit;
  _io : REFERENCE TO HandlingIo;
  _actuator : REFERENCE TO HandlingActuator;
  _fieldbus : REFERENCE TO HandlingFieldbus;
  _axis : REFERENCE TO HandlingAxis;
  _data : REFERENCE TO HandlingDataRef;
  _unit : REFERENCE TO HandlingLinkedUnit;
  _sharedContext : REFERENCE TO SharedContextContainer;
END_VAR

METHOD FB_init : BOOL
VAR_INPUT
  bInitRetains : BOOL; // if TRUE, the retain variables are initialized (warm start / cold start)
  bInCopyCode : BOOL;  // if TRUE, the instance afterwards gets moved into the copy code (online change)
  unit : REFERENCE TO HandlingUnit;
END_VAR
_parent REF= unit;
_alarming := unit._alarming;
_io REF= unit._equipment.Io;
_actuator REF= unit._equipment.Actuator;
_fieldbus REF= unit._equipment.Fieldbus;
_axis REF= unit._equipment.Axis;
_unit REF= unit._equipment.Unit;
_data REF= unit._data;
_loggerDiagnostics.SetLogger(unit._logger);

_sharedContext REF= ZModuleProgram.SharedContext;
END_METHOD

METHOD StepDecoded : ZCore.ZString
VAR_INPUT
  stepIndex : INT;
END_VAR
VAR_INST
  _stepIndexDecoded : HandlingStep;
END_VAR
_stepIndexDecoded := stepIndex;
stepDecoded := TO_STRING(_stepIndexDecoded);
END_METHOD

END_FUNCTION_BLOCK

// ---- ZApp/Unit/Handling/_States/HandlingSequenceAutomatic.TcPOU
FUNCTION_BLOCK HandlingSequenceAutomatic EXTENDS HandlingSequence IMPLEMENTS ZCore.ISequence
VAR
  _step : ZCore.Step(HandlingStep.AutomaticBegin, HandlingStep.AutomaticEnd);
  _timer : ZAux.Timer;
  _rand : ZAux.RandomUniform(seed:=4, low:=1, high:=4);
  
  _speed : LREAL := 100;
  _path : Path1d;
  _newTargetZone, _currentTargetZone : INT;
  _sortedRegions : ARRAY[0..2] OF ZApplication.IRegion;
END_VAR

IF NOT Busy THEN
  RETURN;
END_IF

IF OnStart(_step) THEN
  ; // init custom sequence variables here ...
END_IF

IF OnStop() THEN
  RETURN; // external stop was triggered
END_IF

IF OnHalt() THEN
  Halting := TRUE;
END_IF

REPEAT
  LogStep();

  CASE _step.Index OF
    (* -------------------------------------------------------------------------------------------------------------------------------- *)
    HandlingStep.AutomaticBegin:
    (* -------------------------------------------------------------------------------------------------------------------------------- *)
      IF _step.OnEntry()
      THEN
        ;
      END_IF

      _step.SetNext(HandlingStep.AutomaticWait);
      
    (* -------------------------------------------------------------------------------------------------------------------------------- *)
    HandlingStep.AutomaticWait:
    (* -------------------------------------------------------------------------------------------------------------------------------- *)
      IF _step.OnEntry()
      THEN
        _timer.WaitAsync(0.3);
      END_IF

      IF Halting
      THEN
        _step.SetNext(HandlingStep.AutomaticEnd);
        
      ELSIF _timer.Done
      THEN
      
        WHILE _newTargetZone = _currentTargetZone
        DO
          _newTargetZone := LIMIT(1, LREAL_TO_INT(ZPlatform.Floor(_rand.Next())) , 3); 
        END_WHILE
        
        _currentTargetZone := _newTargetZone;
        _step.SetNext(HandlingStep.AutomaticReservePath);
      END_IF      
    
    (* -------------------------------------------------------------------------------------------------------------------------------- *)    
    HandlingStep.AutomaticReservePath:
    (* -------------------------------------------------------------------------------------------------------------------------------- *)
      IF _step.OnEntry()
      THEN
        _path
          .WithSortedRegions(ADR(_sortedRegions), 3)
          .WithWidth(50)
          .WithSafetyMargin(_speed * 0.01 * 10) // 10 cycles safety margin
          .FromPosition(_axis.AxisX.ActualPosition)
          .ToPosition(TargetPosition(_currentTargetZone))
          .ReserveAsync(_parent);          
      END_IF
      
      _path.Cyclic();

      Await(_path, HandlingStep.AutomaticMoveThroughRegion); 
    
    (* -------------------------------------------------------------------------------------------------------------------------------- *)    
    HandlingStep. AutomaticMoveThroughRegion:
    (* -------------------------------------------------------------------------------------------------------------------------------- *)    
      IF _step.OnEntry()
      THEN
        _axis.AxisX.MoveAbsoluteAsync(THIS^, _path.CurrentEdge, _speed);
      END_IF
      
      IF _path.RegionsToPass = 0
      THEN
        _step.SetNext(HandlingStep.AutomaticMoveToEndPosition);
      ELSIF _path.CheckAndLock(_axis.AxisX.ActualPosition)
      THEN
        _path.IncrementRegion(); 
        _step.SetNext(HandlingStep.AutomaticMoveThroughRegion);
      END_IF

      Assert(_axis.AxisX);
        
    (* -------------------------------------------------------------------------------------------------------------------------------- *)
    HandlingStep.AutomaticMoveToEndPosition:
    (* -------------------------------------------------------------------------------------------------------------------------------- *)
      IF _step.OnEntry()
      THEN
        _axis.AxisX.MoveAbsoluteAsync(THIS^, position := TargetPosition(_currentTargetZone), speed := _speed);
      END_IF
      
      Await(obj1:=_axis.AxisX, nextStep:=HandlingStep.AutomaticWait);
    
    (* -------------------------------------------------------------------------------------------------------------------------------- *)
    HandlingStep.AutomaticEnd:
    (* -------------------------------------------------------------------------------------------------------------------------------- *)
      SetBusy(FALSE);
  
  ELSE
    Abort('sequence contains unhandled step');
  END_CASE
UNTIL _step.IsNotRepeatable() OR_ELSE NOT Busy END_REPEAT

METHOD TargetPosition : LREAL
VAR_INPUT
  zone : INT;
END_VAR
CASE zone
OF
  1: TargetPosition := 50;
  2: TargetPosition := 200;
  3: TargetPosition := 400;  
END_CASE
END_METHOD

END_FUNCTION_BLOCK

// ---- ZApp/Unit/Handling/_States/Path1d.TcPOU
FUNCTION_BLOCK Path1d EXTENDS ZCore.Object IMPLEMENTS IPathQuery, IPathQuery2, IPathQuery3, ZCore.IUnmanagedObject
VAR
  _owner : REFERENCE TO Unit;
  _fromPosition, _toPosition : LREAL;
  _direction : INT;
  _halfWidth, _safetyMargin : LREAL;
  _regions : POINTER TO ZApplication.Region;
  _regionEnd : INT;
  
  _maxRegions : DINT := 5;
  _regionIndicesBuffer : ARRAY[0..5] OF INT;
  _regionIndices : ZCore.RingBufferInt(_maxRegions, ADR(_regionIndicesBuffer));
END_VAR

METHOD CheckAndLock : BOOL;
VAR_INPUT
  pos : LREAL;
END_VAR
VAR_INST
  region : REFERENCE TO ZApplication.Region;
  corner1WithMargin, corner2WithMargin : Vector4;
END_VAR
IF _regionIndices.Empty
THEN
  CheckAndLock := TRUE;
  RETURN;
END_IF

region REF= _regions[_regionIndices.ItemAt(0)];

corner1WithMargin.X := pos - _halfWidth - _safetyMargin;
corner2WithMargin.X := pos + _halfWidth + _safetyMargin;

CheckAndLock := 
  region.IntersectsAABB(corner1WithMargin, corner2WithMargin) AND_THEN
  region.TryLock(_owner);
END_METHOD

PROPERTY CurrentEdge : LREAL
GET
IF _regionIndices.Empty
THEN
  CurrentEdge := _toPosition;
  RETURN;
END_IF

IF _direction < 0
THEN
  CurrentEdge := _regions[_regionIndices.ItemAt(0)].Corner2.X + _halfWidth;
ELSE
  CurrentEdge := _regions[_regionIndices.ItemAt(0)].Corner1.X - _halfWidth;
END_IF
END_GET
END_PROPERTY

METHOD Cyclic
IF NOT Busy
THEN
  RETURN;
END_IF
END_METHOD

METHOD FromPosition : IPathQuery2
VAR_INPUT
  pos : LREAL;
END_VAR
_fromPosition := pos;

FromPosition := THIS^;
END_METHOD

METHOD IncrementRegion
VAR_INST
  intervalMin : LREAL;
  intervalMax : LREAL;
  i : INT;
  
  corner1, corner2 : Vector4;
END_VAR
IF NOT _regionIndices.Empty
THEN
  _regionIndices.PopFirstItem();
END_IF
END_METHOD

PROPERTY RegionsToPass : DINT
GET
RegionsToPass := _regionIndices.Size;
END_GET
END_PROPERTY

METHOD ReserveAsync
VAR_INPUT
  unit : REFERENCE TO Unit;
END_VAR
VAR_INST
  intervalMin : LREAL;
  intervalMax : LREAL;
  i : INT;
  
  corner1, corner2 : Vector4;
END_VAR
intervalMin := MIN(_fromPosition - _halfWidth, _toPosition - _halfWidth);
intervalMax := MAX(_fromPosition + _halfWidth, _toPosition + _halfWidth);

_owner REF= unit;
_direction := SEL(_fromPosition < _toPosition, 1, -1);

corner1.X := intervalMin;
corner2.X := intervalMax;

_regionIndices.Clear();
FOR i := 0 TO _regionEnd BY _direction
DO
  IF _regions[i].IntersectsAABB(corner1, corner2)
  THEN
    _regionIndices.Append(i);
  END_IF
END_FOR

SetBusy(TRUE);
END_METHOD

METHOD ToPosition : IPathQuery3
VAR_INPUT
  pos : LREAL;
END_VAR
_toPosition := pos;
END_METHOD

METHOD WithSafetyMargin : IPathQuery
VAR_INPUT
  margin : LREAL;
END_VAR
_safetyMargin := margin;

WithSafetyMargin := THIS^;
END_METHOD

METHOD WithSortedRegions : IPathQuery
VAR_INPUT
  regions : POINTER TO ZApplication.Region;
  regionCount : INT;
END_VAR
_regions := regions;
_regionEnd := regionCount-1;

WithSortedRegions := THIS^;
END_METHOD

METHOD WithWidth : IPathQuery
VAR_INPUT
  width : LREAL;
END_VAR
_halfWidth := width * 0.5;

WithWidth := THIS^;
END_METHOD

END_FUNCTION_BLOCK

// ---- ZApp/Unit/Handling/_States/HandlingSequenceStop.TcPOU
FUNCTION_BLOCK HandlingSequenceStop EXTENDS HandlingSequence IMPLEMENTS ZCore.ISequence
VAR
  _step : ZCore.Step(HandlingStep.StopBegin, HandlingStep.StopEnd);
  _timerSim : ZAux.Timer;
END_VAR

IF OnStart(_step) THEN
  ; // init custom sequence variables here ...
END_IF

REPEAT
  LogStep();

  CASE _step.Index OF
    (* -------------------------------------------------------------------------------------------------------------------------------- *)
    HandlingStep.StopBegin:
    (* -------------------------------------------------------------------------------------------------------------------------------- *)
      IF _step.OnEntry()
      THEN
        _timerSim.WaitAsync(5);
			END_IF
      
      Await(_timerSim, nextStep:=HandlingStep.StopEnd);
      // _step.SetNext(index:=HandlingStep.StopEnd);

    (* -------------------------------------------------------------------------------------------------------------------------------- *)
    HandlingStep.StopEnd:
    (* -------------------------------------------------------------------------------------------------------------------------------- *)    
      SetBusy(FALSE);
  
  ELSE
    Abort('sequence contains unhandled step');
  END_CASE
UNTIL _step.IsNotRepeatable() OR_ELSE NOT Busy END_REPEAT

END_FUNCTION_BLOCK

// ---- ZApp/Unit/Handling/_States/HandlingSequenceGoHome.TcPOU
FUNCTION_BLOCK HandlingSequenceGoHome EXTENDS HandlingSequence IMPLEMENTS ZCore.ISequence
VAR
  _step : ZCore.Step(HandlingStep.GohomeBegin, HandlingStep.GohomeEnd);
  _timer : ZAux.Timer;
END_VAR

IF NOT Busy THEN
  RETURN;
END_IF

IF OnStart(_step) THEN
  ; // init custom sequence variables here ...
END_IF

IF OnStop() THEN
  RETURN; // external stop was triggered
END_IF

IF OnHalt() THEN
  ; // Halting := TRUE; // Uncomment to acknowledge that the sequence is halting
END_IF

REPEAT
  LogStep();

  CASE _step.Index OF
    (* -------------------------------------------------------------------------------------------------------------------------------- *)
    HandlingStep.GoHomeBegin:
    (* -------------------------------------------------------------------------------------------------------------------------------- *)
      IF _step.OnEntry()
      THEN
        _timer.WaitAsync(2);
			END_IF
      
      Await(_timer, nextStep:=HandlingStep.GoHomeEnd);
      // _step.SetNext(index:=HandlingStep.GoHomeEnd);

    (* -------------------------------------------------------------------------------------------------------------------------------- *)
    HandlingStep.GoHomeEnd:
    (* -------------------------------------------------------------------------------------------------------------------------------- *)
      SetBusy(FALSE);
  
  ELSE
    Abort('sequence contains unhandled step');
  END_CASE
UNTIL _step.IsNotRepeatable() OR_ELSE NOT Busy END_REPEAT

END_FUNCTION_BLOCK

// ---- ZApp/Unit/Handling/_States/HandlingSequenceFaultReaction.TcPOU
FUNCTION_BLOCK HandlingSequenceFaultReaction EXTENDS HandlingSequence IMPLEMENTS ZCore.ISequence
VAR
  _step : ZCore.Step(HandlingStep.FaultReactionBegin, HandlingStep.FaultReactionEnd);
  _timerSim : ZAux.Timer;
END_VAR

IF OnStart(_step) THEN
  ; // init custom sequence variables here ...
END_IF

REPEAT
  LogStep();

  CASE _step.Index OF
    (* -------------------------------------------------------------------------------------------------------------------------------- *)
    HandlingStep.FaultReactionBegin:
    (* -------------------------------------------------------------------------------------------------------------------------------- *)
      IF _step.OnEntry()
      THEN
        _timerSim.WaitAsync(5);
			END_IF
      
      Await(_timerSim, nextStep:=HandlingStep.FaultReactionEnd);
      // _step.SetNext(index:=HandlingStep.FaultReactionEnd);

    (* -------------------------------------------------------------------------------------------------------------------------------- *)
    HandlingStep.FaultReactionEnd:
    (* -------------------------------------------------------------------------------------------------------------------------------- *)    
      SetBusy(FALSE);
  
  ELSE
    Abort('sequence contains unhandled step');
  END_CASE
UNTIL _step.IsNotRepeatable() OR_ELSE NOT Busy END_REPEAT

END_FUNCTION_BLOCK

// ---- ZApp/Unit/Handling/HandlingUnitProgram.TcPOU
/// each unit can run in its own PROGRAM and Task, respectively. However, this is optional and one may also
/// instantiate the unit in the ModuleProgram.
/// In order to keep initialization to a minimum, all ModuleContext objects that are required by the Unit are
/// given as FB_init parameter. These objects are
/// * data structs
/// * communication structs
/// * busmaster(s)
/// A unit should always be a root object (no parent) if it is running in its own context. If it runs in the same
/// task as the Module the parent may be set to the Module's Application.
PROGRAM HandlingUnitProgram
VAR
{region "Handling1"}
{undefine RunInSeparateProgram}
{IF NOT (defined (Handling1_disabled)) AND (defined (RunInSeparateProgram))}
  Handling1 : HandlingUnit(displayName := 'Handling1', // name of the unit (for logging)
    parent:= 0,
    configdata := ZGlobal.Data.Config.Handling1,
    machinedata := ZGlobal.Data.Machine.Handling1,
    calibrationdata := ZGlobal.Data.Calibration.Handling1,
    com := ZGlobal.Com.Unit.Handling1,
    logger := Logger,
    alarming:= Alarming);
  {attribute 'section' := '__ZwPlcUnitProgramDeclaration__'}
  {attribute 'ZId' := 'daa053b3-ae33-4567-9b11-72e6fc346262'}
{END_IF}
{endregion}
{region "Handling2"}
{undefine RunInSeparateProgram}
{IF NOT (defined (Handling2_disabled)) AND (defined (RunInSeparateProgram))}
  Handling2 : HandlingUnit(displayName := 'Handling2', // name of the unit (for logging)
    parent:= 0,
    configdata := ZGlobal.Data.Config.Handling2,
    machinedata := ZGlobal.Data.Machine.Handling2,
    calibrationdata := ZGlobal.Data.Calibration.Handling2,
    com := ZGlobal.Com.Unit.Handling2,
    logger := Logger,
    alarming:= Alarming);
  {attribute 'section' := '__ZwPlcUnitProgramDeclaration__'}
  {attribute 'ZId' := '686d4019-fd8f-49d1-bfb7-e2c5e589b8a3'}
{END_IF}
{endregion}
{region "Handling3"}
{undefine RunInSeparateProgram}
{IF NOT (defined (Handling3_disabled)) AND (defined (RunInSeparateProgram))}
  Handling3 : HandlingUnit(displayName := 'Handling3', // name of the unit (for logging)
    parent:= 0,
    configdata := ZGlobal.Data.Config.Handling3,
    machinedata := ZGlobal.Data.Machine.Handling3,
    calibrationdata := ZGlobal.Data.Calibration.Handling3,
    com := ZGlobal.Com.Unit.Handling3,
    logger := Logger,
    alarming:= Alarming);
  {attribute 'section' := '__ZwPlcUnitProgramDeclaration__'}
  {attribute 'ZId' := '12b42cce-14ce-45ff-90cd-901aacabced4'}
{END_IF}
{endregion}
{region "Handling4"}
{undefine RunInSeparateProgram}
{IF NOT (defined (Handling4_disabled)) AND (defined (RunInSeparateProgram))}
  Handling4 : HandlingUnit(displayName := 'Handling4', // name of the unit (for logging)
    parent:= 0,
    configdata := ZGlobal.Data.Config.Handling4,
    machinedata := ZGlobal.Data.Machine.Handling4,
    calibrationdata := ZGlobal.Data.Calibration.Handling4,
    com := ZGlobal.Com.Unit.Handling4,
    logger := Logger,
    alarming:= Alarming);
  {attribute 'section' := '__ZwPlcUnitProgramDeclaration__'}
  {attribute 'ZId' := '0a2dd986-966c-44be-a2b7-029bd083f361'}
{END_IF}
{endregion}
{attribute '__ZwPlcUnitProgramDeclaration__'} // Do not remove this attribute! It is used for code generation.
END_VAR

// run the unit - the cylics of all children will be called as well

{region "Handling1"}
{undefine RunInSeparateProgram}
{IF NOT (defined (Handling1_disabled)) AND (defined (RunInSeparateProgram))}
  Handling1.Cyclic();
  {attribute 'section' := '__ZwPlcUnitProgramImplementation__'}
  {attribute 'ZId' := 'daa053b3-ae33-4567-9b11-72e6fc346262'}
{END_IF}
{endregion}
{region "Handling2"}
{undefine RunInSeparateProgram}
{IF NOT (defined (Handling2_disabled)) AND (defined (RunInSeparateProgram))}
  Handling2.Cyclic();
  {attribute 'section' := '__ZwPlcUnitProgramImplementation__'}
  {attribute 'ZId' := '686d4019-fd8f-49d1-bfb7-e2c5e589b8a3'}
{END_IF}
{endregion}
{region "Handling3"}
{undefine RunInSeparateProgram}
{IF NOT (defined (Handling3_disabled)) AND (defined (RunInSeparateProgram))}
  Handling3.Cyclic();
  {attribute 'section' := '__ZwPlcUnitProgramImplementation__'}
  {attribute 'ZId' := '12b42cce-14ce-45ff-90cd-901aacabced4'}
{END_IF}
{endregion}
{region "Handling4"}
{undefine RunInSeparateProgram}
{IF NOT (defined (Handling4_disabled)) AND (defined (RunInSeparateProgram))}
  Handling4.Cyclic();
  {attribute 'section' := '__ZwPlcUnitProgramImplementation__'}
  {attribute 'ZId' := '0a2dd986-966c-44be-a2b7-029bd083f361'}
{END_IF}
{endregion}
{attribute '__ZwPlcUnitProgramImplementation__'} // Do not remove this attribute! It is used for code generation.

END_PROGRAM
